ORGANIZATION_BLOCK MAIN
{ S7_Optimized_Access := 'false' }
    VAR_TEMP
        lastTimerValue: TIME;
        curDeltaTime: TIME;
        curDeltaSecs: REAL;
        state1: STATE;
        progress: BOOL;
        loopCount: INT;
        b1: BOOL;
        b2: BOOL;
        timerValue0: TIME;
        timerValue1: TIME;
    END_VAR

BEGIN

    // Handle 'time' and cycle time.
    "DB".cnt := "DB".cnt + 1;

    timer0.TON(IN := "DB".curTimer = 0, PT := T#1D);
    timer1.TON(IN := "DB".curTimer = 1, PT := T#1D);
    timerValue0 := timer0.ET;
    timerValue1 := timer1.ET;

    lastTimerValue := "DB".curTimerValue;
    IF "DB".curTimer = 0 THEN
        "DB".curTimerValue := timerValue0;
    ELSE
        "DB".curTimerValue := timerValue1;
    END_IF;
    curDeltaTime := "DB".curTimerValue - lastTimerValue;
    curDeltaSecs := DINT_TO_REAL(TIME_TO_DINT(curDeltaTime)) / 1000;
    "DB".curTime := "DB".curTime + curDeltaSecs;

    IF "DB".cnt MOD 10 = 0 THEN
        "DB".curTimer := 1 - "DB".curTimer;
        "DB".curTimerValue := T#0S;
        timer0.TON(IN := "DB".curTimer = 0, PT := T#1D);
        timer1.TON(IN := "DB".curTimer = 1, PT := T#1D);
        timerValue0 := timer0.ET;
        timerValue1 := timer1.ET;
    END_IF;

    IF "DB".first THEN
        "DB".first := FALSE;

        // Initialize state variables for initial state.
        "DB".state0.dvar_M_hw_button := 4;
        "DB".state0.dvar_M_hw_lamp_bit := FALSE;
        "DB".state0.dvar_M_hw_lamp := 1;
        "DB".state0.dvar_M_sup := 6;
        "DB".state0.cvar_M_timer_t := 0.0;
        "DB".state0.dvar_M_timer := 0;
    ELSE
        // Update continuous variables for time delay.
        state1.cvar_M_timer_t := "DB".state0.cvar_M_timer_t + curDeltaSecs * derivcvar_M_timer_t("DB".state0);

        "DB".state0.curTime := "DB".curTime;
        "DB".state0.cvar_M_timer_t := state1.cvar_M_timer_t;
    END_IF;

    // Event loop.
    WHILE TRUE DO
        progress := FALSE;

        // Event "button.push".
        IF NOT progress THEN
            b1 := ("DB".state0.dvar_M_hw_button) = (4);
            b1 := b1 AND (ivar_hw_button_bit);
            IF b1 THEN
                b2 := ("DB".state0.dvar_M_sup) = (6);
                b2 := b2 OR (("DB".state0.dvar_M_sup) = (10));
                b2 := b2 OR (("DB".state0.dvar_M_sup) = (11));
                b2 := b2 OR (("DB".state0.dvar_M_sup) = (13));
                b2 := b2 OR (("DB".state0.dvar_M_sup) = (15));
                b1 := b1 AND (b2);
            END_IF;
            IF b1 THEN
                progress := TRUE;
                state1 := "DB".state0;

                state1.dvar_M_hw_button := 3;
                IF (("DB".state0.dvar_M_sup) = (6)) THEN
                    state1.dvar_M_sup := 8;
                ELSIF (("DB".state0.dvar_M_sup) = (10)) THEN
                    state1.dvar_M_sup := 8;
                ELSIF (("DB".state0.dvar_M_sup) = (11)) THEN
                    state1.dvar_M_sup := 9;
                ELSIF (("DB".state0.dvar_M_sup) = (13)) THEN
                    state1.dvar_M_sup := 12;
                ELSIF (("DB".state0.dvar_M_sup) = (15)) THEN
                    state1.dvar_M_sup := 14;
                END_IF;

                "DB".state0 := state1;
            END_IF;
        END_IF;

        // Event "button.release".
        IF NOT progress THEN
            b1 := ("DB".state0.dvar_M_hw_button) = (3);
            b1 := b1 AND (NOT(ivar_hw_button_bit));
            IF b1 THEN
                b2 := ("DB".state0.dvar_M_sup) = (8);
                b2 := b2 OR (("DB".state0.dvar_M_sup) = (9));
                b2 := b2 OR (("DB".state0.dvar_M_sup) = (12));
                b2 := b2 OR (("DB".state0.dvar_M_sup) = (14));
                b2 := b2 OR (("DB".state0.dvar_M_sup) = (7));
                b1 := b1 AND (b2);
            END_IF;
            IF b1 THEN
                progress := TRUE;
                state1 := "DB".state0;

                state1.dvar_M_hw_button := 4;
                IF (("DB".state0.dvar_M_sup) = (8)) THEN
                    state1.dvar_M_sup := 10;
                ELSIF (("DB".state0.dvar_M_sup) = (9)) THEN
                    state1.dvar_M_sup := 11;
                ELSIF (("DB".state0.dvar_M_sup) = (12)) THEN
                    state1.dvar_M_sup := 13;
                ELSIF (("DB".state0.dvar_M_sup) = (14)) THEN
                    state1.dvar_M_sup := 15;
                ELSIF (("DB".state0.dvar_M_sup) = (7)) THEN
                    state1.dvar_M_sup := 6;
                END_IF;

                "DB".state0 := state1;
            END_IF;
        END_IF;

        // Event "lamp.off".
        IF NOT progress THEN
            b1 := ("DB".state0.dvar_M_hw_lamp) = (2);
            IF b1 THEN
                b2 := ("DB".state0.dvar_M_sup) = (14);
                b2 := b2 OR (("DB".state0.dvar_M_sup) = (15));
                b1 := b1 AND (b2);
            END_IF;
            IF b1 THEN
                progress := TRUE;
                state1 := "DB".state0;

                state1.dvar_M_hw_lamp_bit := FALSE;
                state1.dvar_M_hw_lamp := 1;
                IF (("DB".state0.dvar_M_sup) = (14)) THEN
                    state1.dvar_M_sup := 7;
                ELSIF (("DB".state0.dvar_M_sup) = (15)) THEN
                    state1.dvar_M_sup := 6;
                END_IF;

                "DB".state0 := state1;
            END_IF;
        END_IF;

        // Event "lamp.on".
        IF NOT progress THEN
            b1 := ("DB".state0.dvar_M_hw_lamp) = (1);
            IF b1 THEN
                b2 := ("DB".state0.dvar_M_sup) = (8);
                b2 := b2 OR (("DB".state0.dvar_M_sup) = (10));
                b1 := b1 AND (b2);
            END_IF;
            IF b1 THEN
                progress := TRUE;
                state1 := "DB".state0;

                state1.dvar_M_hw_lamp_bit := TRUE;
                state1.dvar_M_hw_lamp := 2;
                IF (("DB".state0.dvar_M_sup) = (8)) THEN
                    state1.dvar_M_sup := 9;
                ELSIF (("DB".state0.dvar_M_sup) = (10)) THEN
                    state1.dvar_M_sup := 11;
                END_IF;

                "DB".state0 := state1;
            END_IF;
        END_IF;

        // Event "timer.start".
        IF NOT progress THEN
            b2 := ("DB".state0.dvar_M_sup) = (9);
            b2 := b2 OR (("DB".state0.dvar_M_sup) = (11));
            b1 := b2;
            b1 := b1 AND (("DB".state0.dvar_M_timer) = (0));
            IF b1 THEN
                progress := TRUE;
                state1 := "DB".state0;

                IF (("DB".state0.dvar_M_sup) = (9)) THEN
                    state1.dvar_M_sup := 12;
                ELSIF (("DB".state0.dvar_M_sup) = (11)) THEN
                    state1.dvar_M_sup := 13;
                END_IF;
                state1.cvar_M_timer_t := 0.0;
                state1.dvar_M_timer := 5;

                "DB".state0 := state1;
            END_IF;
        END_IF;

        // Event "timer.timeout".
        IF NOT progress THEN
            b2 := ("DB".state0.dvar_M_sup) = (12);
            b2 := b2 OR (("DB".state0.dvar_M_sup) = (13));
            b1 := b2;
            b1 := b1 AND (("DB".state0.dvar_M_timer) = (5));
            b1 := b1 AND (("DB".state0.cvar_M_timer_t) >= (3.0));
            IF b1 THEN
                progress := TRUE;
                state1 := "DB".state0;

                IF (("DB".state0.dvar_M_sup) = (12)) THEN
                    state1.dvar_M_sup := 14;
                ELSIF (("DB".state0.dvar_M_sup) = (13)) THEN
                    state1.dvar_M_sup := 15;
                END_IF;
                state1.dvar_M_timer := 0;

                "DB".state0 := state1;
            END_IF;
        END_IF;

        // Done with events?
        IF NOT progress THEN
            EXIT;
        END_IF;

        // Protect against events that are always enabled.
        loopCount := loopCount + 1;
        IF loopCount >= 100 THEN
            "DB".loopsKilled := "DB".loopsKilled + 1;
            EXIT;
        END_IF;
    END_WHILE;
END_ORGANIZATION_BLOCK
